SUBAPPLICATION Uebung_001c (* DigitalInput_I1 auf DigitalOutput_Q1 --> Eingang abfragen bei Boot. *)
  (* Standard: 61499-2; Description: Copyright (c) 2023 Meisterschulen am Ostbahnhof This program and the accompanying materials are made available under the terms of the Eclipse Public License 2.0 which is available at https://www.eclipse.org/legal/epl-2.0/ SPDX-License-Identifier: EPL-2.0 *)
  (* Version 1.0, 2023-10-23, Franz Höpfinger, Meisterschulen am Ostbahnhof *)
  IMPORT logiBUS::io::DI::logiBUS_DI::Input_I1;
  IMPORT logiBUS::io::DQ::logiBUS_DO::Output_Q1;
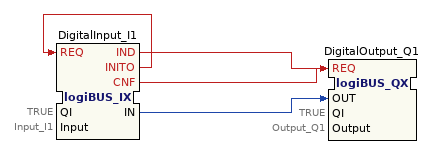
  FBS
    DigitalOutput_Q1 : logiBUS::io::DQ::logiBUS_QX(QI := TRUE, Output := Output_Q1);
    DigitalInput_I1 : logiBUS::io::DI::logiBUS_IX(QI := TRUE, Input := Input_I1);
  END_FBS
  EVENT_CONNECTIONS
    DigitalInput_I1.IND TO DigitalOutput_Q1.REQ;
    DigitalInput_I1.INITO TO DigitalInput_I1.REQ;
    DigitalInput_I1.CNF TO DigitalOutput_Q1.REQ;
  END_CONNECTIONS
  DATA_CONNECTIONS
    DigitalInput_I1.IN TO DigitalOutput_Q1.OUT;
  END_CONNECTIONS
END_SUBAPPLICATION
